// ---- VISUs/Pages/Initializing/InitializingTrayfeederInterupted.TcVIS
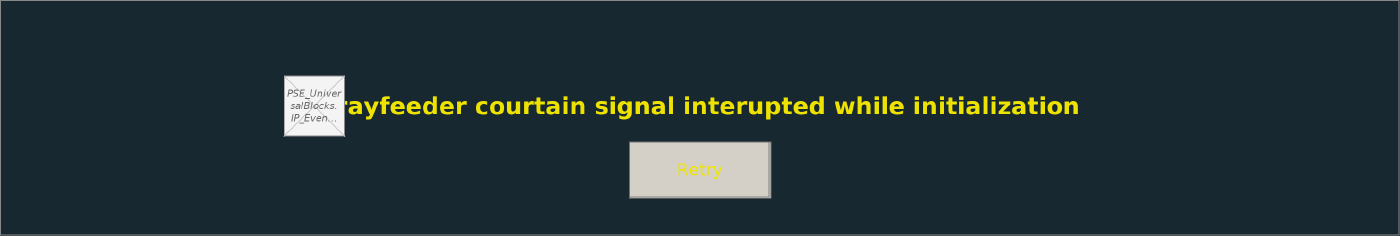
VISUALIZATION InitializingTrayfeederInterupted  // 1480x250
VAR_IN_OUT
	btnTrayfeederInitRetry : BOOL;
END_VAR
    Label (0,92 1480x40), "Trayfeeder courtain signal interupted while initialization"
    Image (300,80 64x64), image: PSE_UniversalBlocks.IP_EventSeverity.error
    Button (665,150 150x60), "Retry"
        toggle btnTrayfeederInitRetry
END_VISUALIZATION

// ---- VISUs/Pages/Initializing/PageInitializing.TcVIS
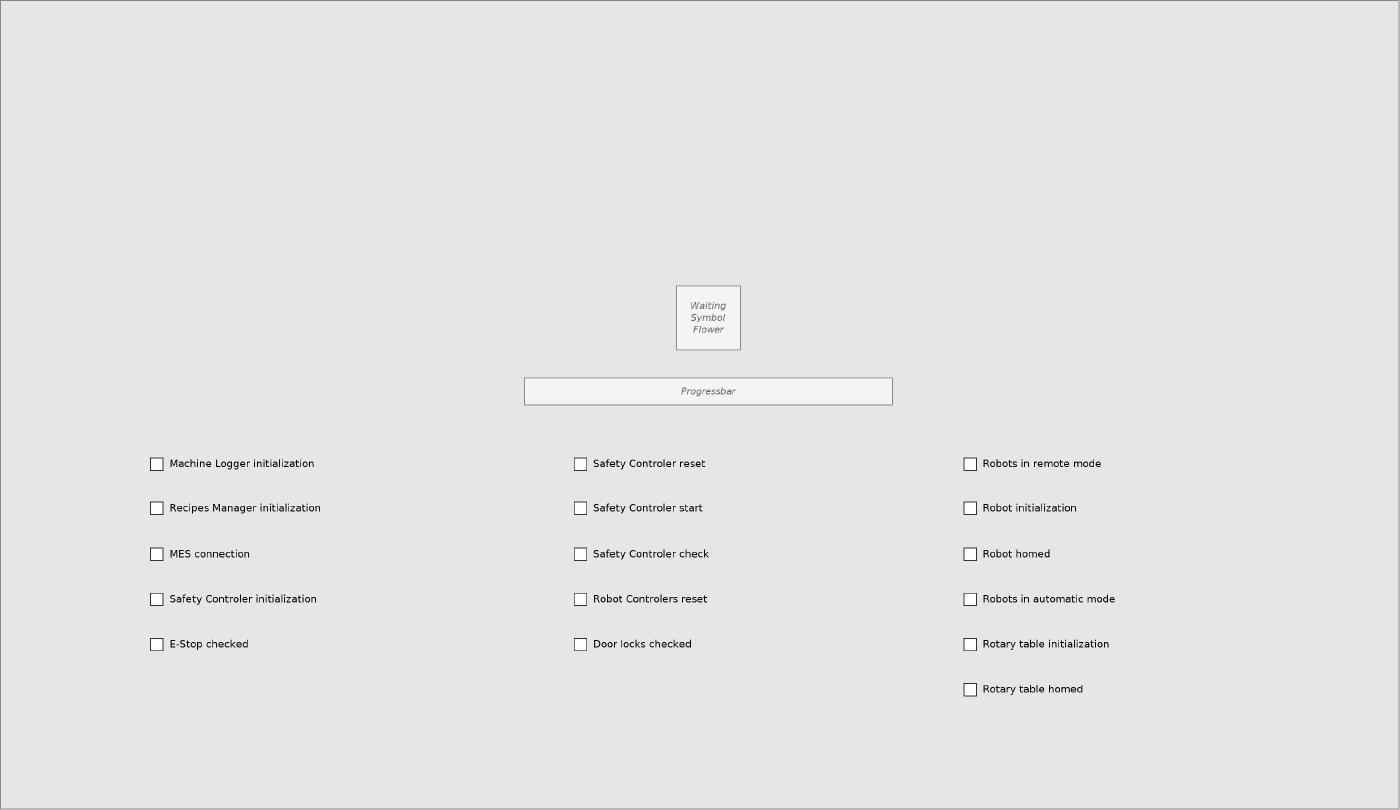
VISUALIZATION PageInitializing  // 1520x880
VAR_IN_OUT
	iProgressBar : USINT;
END_VAR
    Progressbar (569,410 400x30), variable: iProgressBar
    WaitingSymbolFlower (734,310 70x70)
    Checkbox (161,489 300x30), "Machine Logger initialization", variable: PRG_VisuControl.fbVisuControl.stInitializingFrame.bMachineLoggerInitialized, input disabled if: FALSE
    Checkbox (621,636 320x30), "Robot Controlers reset", variable: PRG_VisuControl.fbVisuControl.stInitializingFrame.bRobotControlersResetDone
    Checkbox (1044,537 320x30), "Robot initialization", variable: PRG_VisuControl.fbVisuControl.stInitializingFrame.bRobotOneInitialized
    Checkbox (1044,636 300x30), "Robots in automatic mode", variable: PRG_VisuControl.fbVisuControl.stInitializingFrame.bRobotsInAutomaticMode
    Checkbox (1044,587 320x30), "Robot homed", variable: PRG_VisuControl.fbVisuControl.stInitializingFrame.bRobotOneHomed
    Checkbox (161,537 300x30), "Recipes Manager initialization", variable: PRG_VisuControl.fbVisuControl.stInitializingFrame.bRecipesManagerInitialized, input disabled if: FALSE
    Checkbox (161,587 300x30), "MES connection", variable: PRG_VisuControl.fbVisuControl.stInitializingFrame.bMesConnected, input disabled if: FALSE
    Checkbox (161,636 300x30), "Safety Controler initialization", variable: PRG_VisuControl.fbVisuControl.stInitializingFrame.bSafetyInitialization, input disabled if: FALSE
    Checkbox (161,685 300x30), "E-Stop checked", variable: PRG_VisuControl.fbVisuControl.stInitializingFrame.bEStopChecked, input disabled if: FALSE
    Checkbox (621,685 300x30), "Door locks checked", variable: PRG_VisuControl.fbVisuControl.stInitializingFrame.bDoorsLocked, input disabled if: FALSE
    Checkbox (621,489 320x30), "Safety Controler reset", variable: PRG_VisuControl.fbVisuControl.stInitializingFrame.bSafetyReset, input disabled if: FALSE
    Checkbox (621,537 320x30), "Safety Controler start", variable: PRG_VisuControl.fbVisuControl.stInitializingFrame.bSafetyStart, input disabled if: FALSE
    Checkbox (621,587 320x30), "Safety Controler check", variable: PRG_VisuControl.fbVisuControl.stInitializingFrame.bSafetyCheck
    Checkbox (1044,489 320x30), "Robots in remote mode", variable: PRG_VisuControl.fbVisuControl.stInitializingFrame.bRobotsInRemoteMode
    Checkbox (1044,734 208x30), "Rotary table homed"
    Checkbox (1044,685 293x30), "Rotary table initialization"
END_VISUALIZATION

// ---- VISUs/Pages/PageAlarms.TcVIS
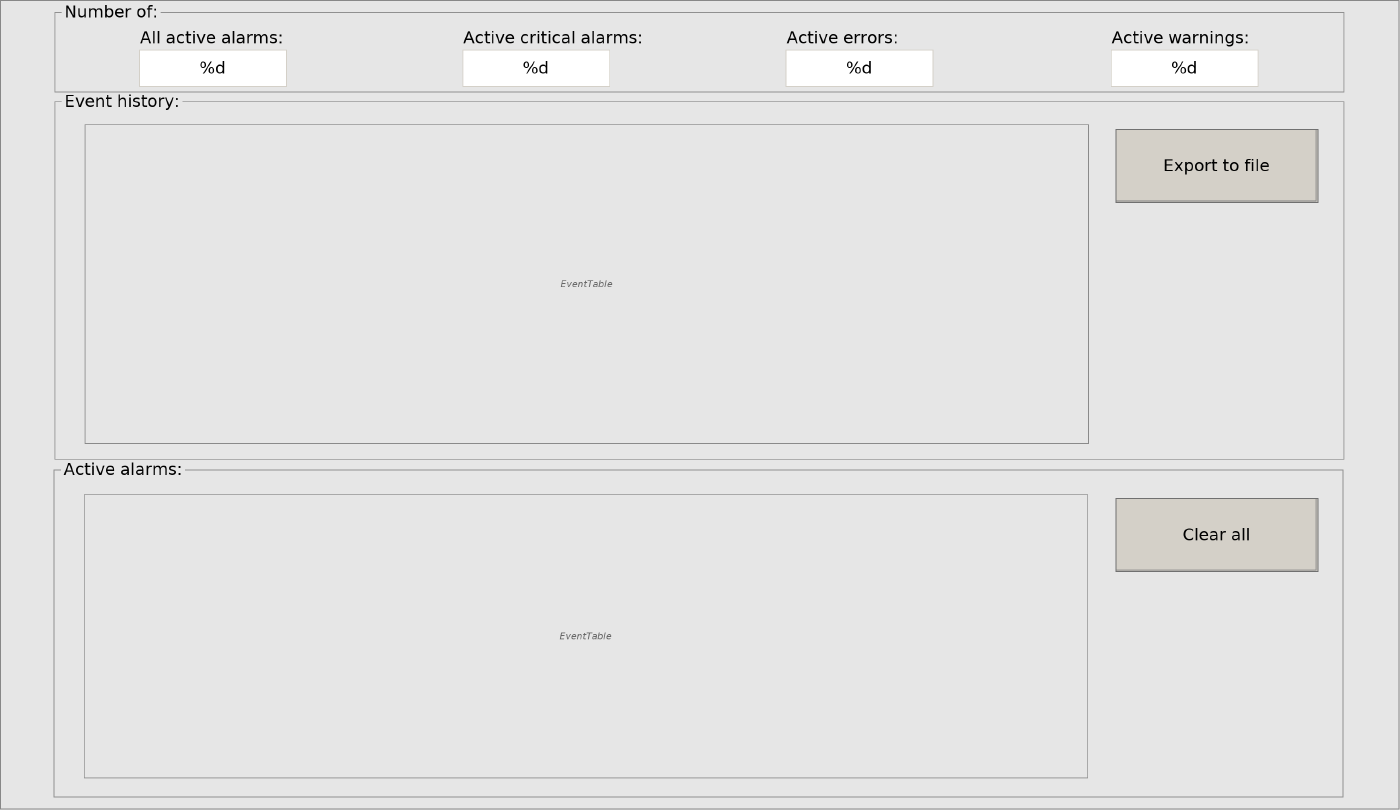
VISUALIZATION PageAlarms  // 1520x880
VAR_IN_OUT
	btnClearAllAlarms 	: BOOL;
	btnExportEvents		: BOOL;
	iActiveAlarms		: UDINT;
	iActiveCritical		: UDINT;
	iActiveErrors		: UDINT;
	iActiveWarrnings	: UDINT;
	arrEvents			: ARRAY[1..iMAX_EVENTS] OF ST_Event;
	arrAlarms			: ARRAY[1..iMAX_EVENTS] OF ST_Event;
END_VAR
    GroupBox (58,502 1400x364), "Active alarms:"
        Frame (33,35 1090x308)
            shows EventTable(data := arrAlarms)
        Button (1153,39 220x80), "Clear all"
            tap btnClearAllAlarms
    GroupBox (59,5 1400x95), "Number of:"
        Label (90,21 210x30), "All active alarms:"
        Textfield (92,49 160x40), "%d", text variable: iActiveAlarms, text list: ''
        Label (441,21 234x30), "Active critical alarms:"
        Textfield (443,49 160x40), "%d", text variable: iActiveCritical, text list: ''
        Label (792,21 210x30), "Active errors:"
        Label (1145,21 210x30), "Active warnings:"
        Textfield (794,49 160x40), "%d", text variable: iActiveErrors, text list: ''
        Textfield (1147,49 160x40), "%d", text variable: iActiveWarrnings, text list: ''
    GroupBox (59,102 1400x397), "Event history:"
        Frame (33,33 1090x347)
            shows EventTable(data := arrEvents)
        Button (1152,38 220x80), "Export to file"
            tap btnExportEvents
END_VISUALIZATION

// ---- VISUs/Pages/Uninitialized/PageUninitialized.TcVIS
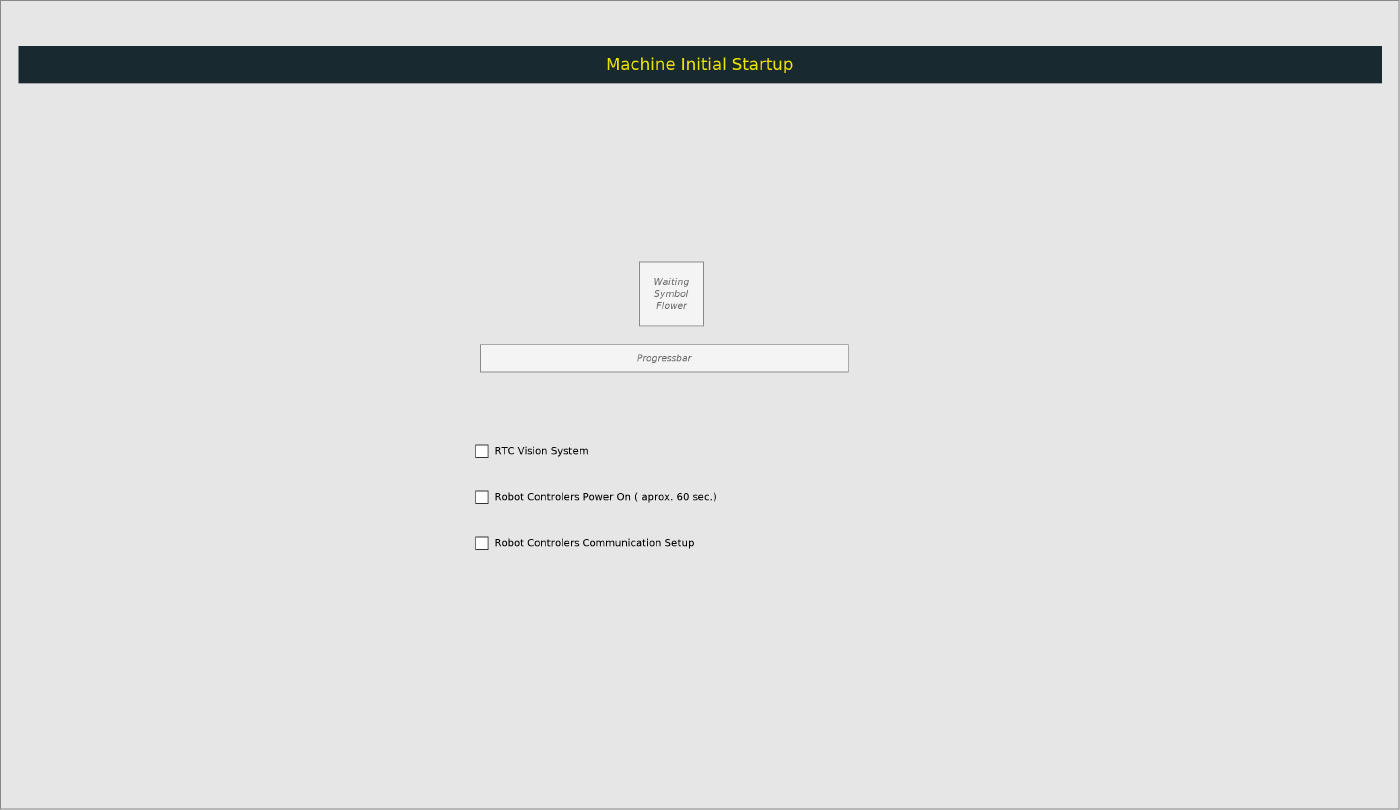
VISUALIZATION PageUninitialized  // 1520x880
    Frame (20,50 1480x780), frame switch variable: PRG_VisuControl.fbVisuControl.eUninitializedFrameSelector
        shows UninitializedStartUpFrame(stUninitializedStartUpFrame := PRG_VisuControl.fbVisuControl.stUninitializedStartUpFrame)
        shows UninitializedSetupFrame()
END_VISUALIZATION

// ---- VISUs/Pages/Uninitialized/UninitializedSetupFrame.TcVIS
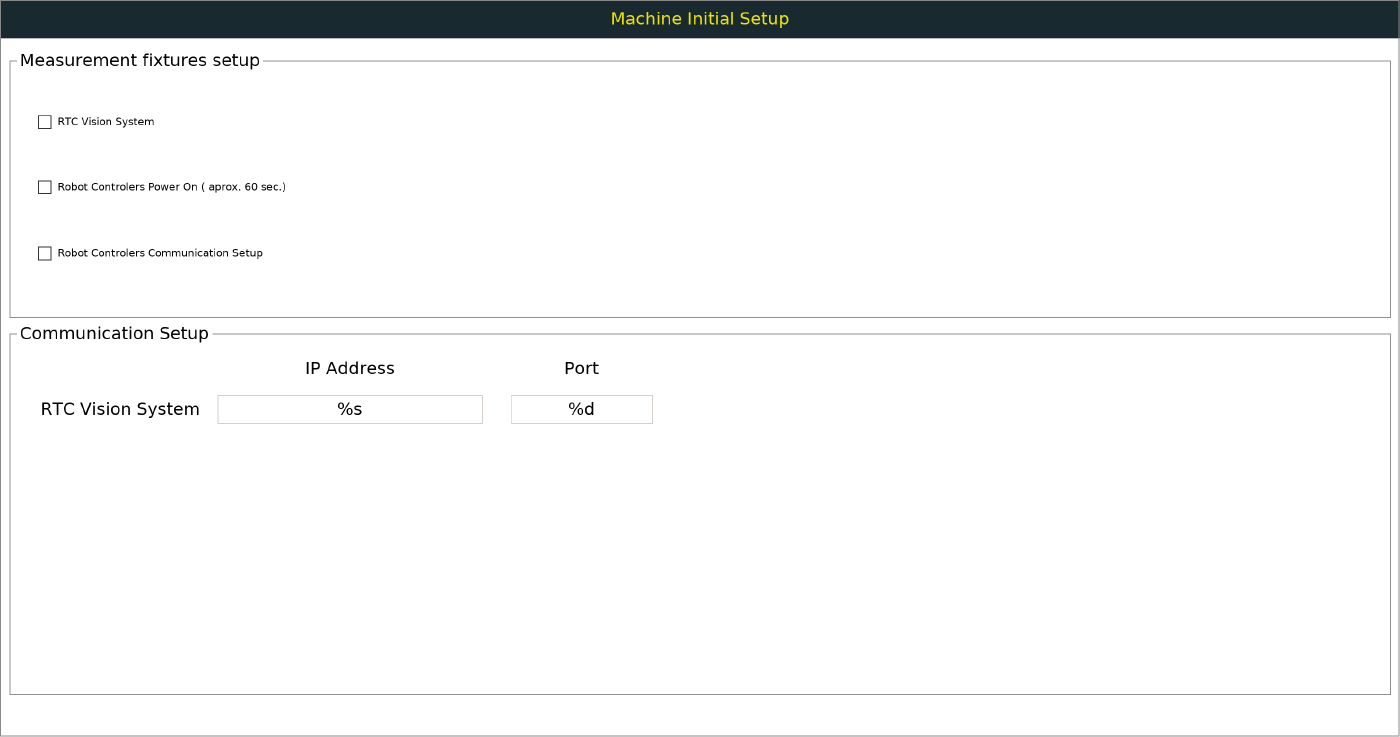
VISUALIZATION UninitializedSetupFrame  // 1480x780
VAR_IN_OUT
	//stUninitializedFrame : ST_UninitializedSetupFrame;
END_VAR
    GroupBox (10,56 1460x280), "Measurement fixtures setup"
        Checkbox (28,58 400x30), "RTC Vision System"
        Checkbox (28,127 450x30), "Robot Controlers Power On ( aprox. 60 sec.)"
        Checkbox (28,197 400x30), "Robot Controlers Communication Setup"
    GroupBox (10,345 1460x390), "Communication Setup"
        Label (30,63 192x50), "RTC Vision System"
        Textfield (220,73 280x30), "%s"
            OnMouseClick: write the text variable via VisuDialogs.Numpad
        Textfield (530,73 150x30), "%d"
            OnMouseClick: write the text variable via VisuDialogs.Numpad
        Label (220,30 280x30), "IP Address"
        Label (530,30 150x30), "Port"
    Rectangle (0,0 1480x40), "Machine Initial Setup"
END_VISUALIZATION

// ---- VISUs/Pages/Uninitialized/UninitializedStartUpFrame.TcVIS
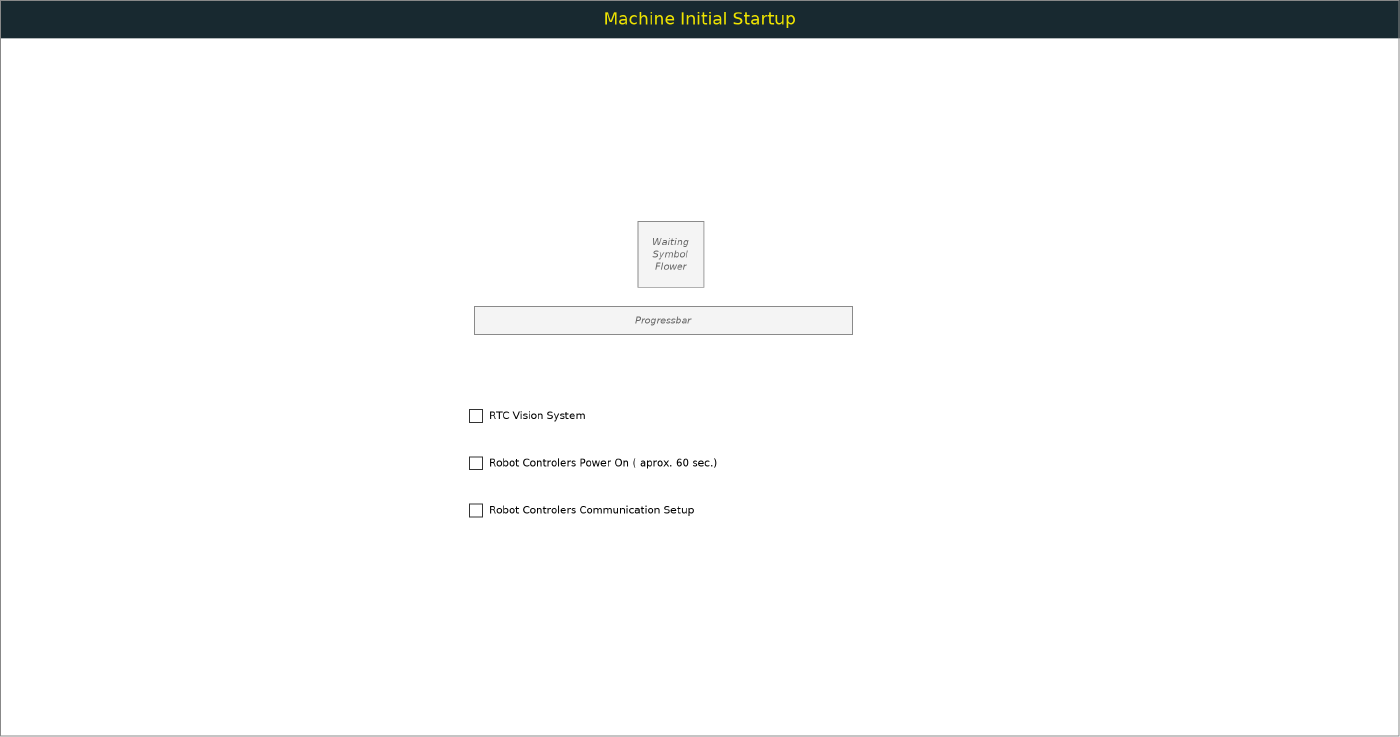
VISUALIZATION UninitializedStartUpFrame  // 1480x780
VAR_IN_OUT
	stUninitializedStartUpFrame	: ST_UninitializedStartUpFrame;
END_VAR
    Rectangle (0,0 1480x40), "Machine Initial Startup"
    Progressbar (501,324 400x30), variable: stUninitializedStartUpFrame.iProgressBar
    Checkbox (494,425 400x30), "RTC Vision System", variable: PRG_VisuControl.fbVisuControl.stUninitializedStartUpFrame.bRTCVisionPowerOn
    Checkbox (494,525 400x30), "Robot Controlers Communication Setup", variable: stUninitializedStartUpFrame.bCR800EtherCatInitialization
    Checkbox (494,475 450x30), "Robot Controlers Power On ( aprox. 60 sec.)", variable: stUninitializedStartUpFrame.bCR800PowerOn
    WaitingSymbolFlower (674,234 70x70)
END_VISUALIZATION
